FUNCTION_BLOCK FB_FeedForwardAuto
VAR_INPUT
	bEnable : BOOL;
	fVelRef : LREAL;
	stOpenLoopSettings : ST_OpenLoopSettings;
END_VAR
VAR_OUTPUT
	fVelFeedFWD : LREAL; 
END_VAR
VAR
	fTempOut : LREAL;
END_VAR

IF fVelRef >= 0.0 THEN
	fTempOut := stOpenLoopSettings.fBoreArea*fVelRef; // Flow to bore side
ELSE
	fTempOut := stOpenLoopSettings.fAnnulusArea * fVelRef;		// FLow to piston side
END_IF

IF bEnable THEN
	fVelFeedFWD := (60000.0*fTempOut)/150.0;
ELSE
	fVelFeedFWD := 0.0;
END_IF

END_FUNCTION_BLOCK

(* stored: Version 1.1.0.1, ProductVersion 3.1.4024.12
   POU FB_FeedForwardAuto: Id {6f66b99a-cf75-432c-82b9-43f8fa7c884e}, SpecialFunc None *)
